Universal Robots PolyScope program: husarion_ext_control.urp

Program husarion_ext_control (installation=default directory=/programs createdIn=5.13.0 lastSavedIn=5.13.0 robotSerialNumber=20185300462)
Calibrated DH parameters: a=[-0.000019, -0.236553, -0.213301, 0.000133, -0.000098, 0]; d=[0.151722, 8.225656, -8.568715, 0.474066, 0.085493, 0.092367]; alpha=[1.570598, -0.007173, -0.0079, 1.57058, -1.572123, 0]; deltaTheta=[0, -0.244422, 0.257137, -0.012712, 0.000041, 0]
InitVariablesNode
Robot Program (runOnlyOnce=false)
  URCap External Control (External Control, FZI Research Center for Information Technology)
Thread Thread_1 (runOnlyOnce=true)
  Script file /programs/husarion_rg2_driver.script
    | modbus_add_signal("10.42.0.49", 255, 16, 3, "joint_out")
    | modbus_add_signal("10.42.0.49", 255, 17, 1, "rg_busy_out")
    | modbus_add_signal("10.42.0.49", 255, 18, 1, "grip_detected_out")
    | 
    | modbus_add_signal("10.42.0.49", 255, 20, 0, "action_trigger_in")
    | modbus_add_signal("10.42.0.49", 255, 128, 2, "joint_in")
    | modbus_add_signal("10.42.0.49", 255, 129, 2, "force_in")
    | 
    | modbus_set_signal_update_frequency("joint_out", 500)
    | modbus_set_signal_update_frequency("rg_busy_out", 500)
    | modbus_set_signal_update_frequency("grip_detected_out", 500)
    | modbus_set_signal_update_frequency("action_trigger_in", 500)
    | modbus_set_signal_update_frequency("joint_in", 500)
    | modbus_set_signal_update_frequency("force_in", 500)
    | 
    | while(True):
    |     if modbus_get_signal_status("action_trigger_in", False):
    |         joint_req = modbus_get_signal_status("joint_in", False) / 10
    |         force_req = modbus_get_signal_status("force_in", False) / 10
    |         rg_grip(joint_req, force_req, 0, False, False)
    |     end
    | 
    |     width = norm(floor(rg_Width * 10))
    |     modbus_set_output_register("joint_out", width, False)
    |     modbus_set_output_signal("rg_busy_out", rg_Busy, False)
    |     modbus_set_output_signal("grip_detected_out", rg_Grip_detected, False)
    | 
    |     sleep(0.05)
    | end
Thread Thread_2 (runOnlyOnce=true)
  Script file /programs/husarion_rg2_watchdog.script
    | modbus_add_signal("10.42.0.49", 255, 19, 1, "watchdog_out")
    | modbus_set_signal_update_frequency("joint_out", 500)
    | 
    | state = False
    | 
    | while(True):
    |     modbus_set_output_signal("watchdog_out", state, False)
    |     state = not state
    |     sleep(0.1)
    | end
